RoboDK station: 29-6-1028.rdk

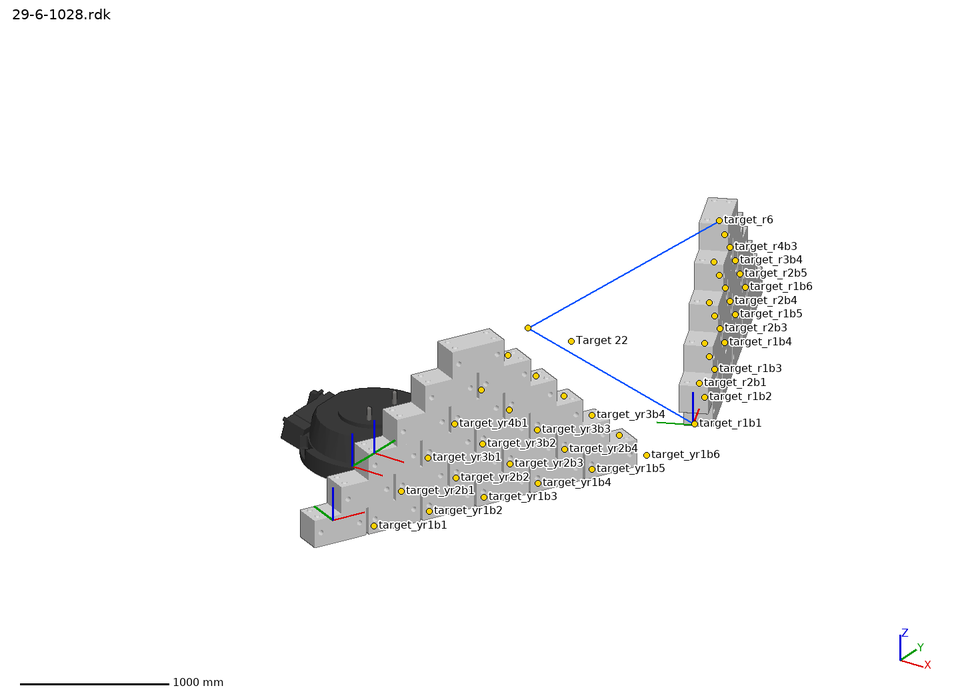
[picture v0: the station drawn from its stored meshes, robots at their saved joint values, targets as dots, program paths as lines]
Station 29-6-1028 (saved by RoboDK 5.4.1). Poses are relative to the parent item; angles as X-Y-Z fixed-axis rotations.
  - folder assets
    - object Floor at (0, 0, 0) mm, size 9000 x 9000 x 0 mm, geometry from Floor.sld
    - object Stairs_v1 at (-2520, 0, 0) mm, size 3922.2 x 7408.9 x 2302 mm, geometry from Stairs_v1.3ds
    - object Frame at (0, 0, 0) mm, size 2000 x 2500 x 199.8 mm, geometry from Frame.stp
  - frame KUKA KR 210-2 Base at (0, 0, 140) mm
    - robot KUKA KR 210-2: 6 axes, payload 210 kg, reach 2700 mm, repeatability 0.06 mm, weight 1267 kg
        joint limits [-185, -146, -119, -350, -125, -350] to [185, 0, 155, 350, 125, 350]; home [0, -128.166, 146.243, 0, -18.127, 0]; saved at [4.205, -124.52, 145.644, 6.755, -21.204, -6.343]
      - tool NEMO_ASM-v2, TCP at (50, 0, 430) mm, size 350 x 350 x 427.5 mm, geometry from NEMO_ASM-v2.stp
    - frame Table 1 at (2403.79, 306.78, 760.01) mm, rotated rx 0 ry 0 rz 115.9 deg
      - target target_r1b1 (Cartesian target) at (-6.3, -11.13, 11.37) mm, rotated rx -176.72 ry 88.61 rz 93.44 deg; joints [-0.522, -50.102, 99.56, 32.766, -52.796, -20.524] of KUKA KR 210-2
      - target target_r1b2 (Cartesian target) at (416.03, -12.09, 10.91) mm, rotated rx -158.93 ry 88.69 rz 112.47 deg; joints [-13.142, -53.707, 107.729, 17.568, -54.069, -9.744] of KUKA KR 210-2
      - target target_r1b3 (Cartesian target) at (839.45, -13.29, 13.06) mm, rotated rx 172.71 ry 89.07 rz 84.11 deg; joints [-27.608, -54.712, 110.113, -0.377, -54.484, 0.097] of KUKA KR 210-2
      - target target_r1b4 (Cartesian target) at (1261.96, -15.87, 12.69) mm, rotated rx 175.27 ry 88.55 rz 86.33 deg; joints [-41.947, -53.093, 105.958, -18.915, -52.906, 11.169] of KUKA KR 210-2
      - target target_r1b5 (Cartesian target) at (1681.19, -17.51, 17.53) mm, rotated rx 170.01 ry 89.31 rz 81.06 deg; joints [-54.307, -48.398, 95.994, -35.345, -52.576, 22.843] of KUKA KR 210-2
      - target target_r1b6 (Cartesian target) at (2102.3, -19.1, 19.95) mm, rotated rx -105.14 ry 89.86 rz 166.05 deg; joints [-64.353, -40.838, 79.979, -50.347, -51.856, 36.8] of KUKA KR 210-2
      - target target_r2b1 (Cartesian target) at (205.96, -10.53, 214.78) mm, rotated rx -150.39 ry 88.9 rz 120.14 deg; joints [-6.706, -59.689, 102.908, 28.081, -45.79, -19.523] of KUKA KR 210-2
      - target target_r2b2 (Cartesian target) at (625.98, -11.98, 212.77) mm, rotated rx -150.6 ry 88.91 rz 119.96 deg; joints [-20.566, -62.512, 108.17, 8.347, -45.007, -5.288] of KUKA KR 210-2
      - target target_r2b3 (Cartesian target) at (1050.36, -15.25, 215.86) mm, rotated rx -170.53 ry 89.44 rz 100.79 deg; joints [-34.887, -61.925, 107.233, -10.832, -45.265, 7.688] of KUKA KR 210-2
      - target target_r2b4 (Cartesian target) at (1470.51, -16.51, 217.48) mm, rotated rx -170.97 ry 89.43 rz 100.55 deg; joints [-48.227, -58.207, 100.325, -29.828, -45.582, 21.741] of KUKA KR 210-2
      - target target_r2b5 (Cartesian target) at (1894.14, -18.95, 219.85) mm, rotated rx -105.55 ry 89.86 rz 166.1 deg; joints [-59.529, -51.207, 87.402, -46.619, -46.767, 36.046] of KUKA KR 210-2
      - target target_r3b1 (Cartesian target) at (413.86, -11.7, 413.85) mm, rotated rx -150.56 ry 88.9 rz 120.16 deg; joints [-13.32, -67.987, 102.857, 22.975, -36.114, -18.141] of KUKA KR 210-2
      - target target_r3b2 (Cartesian target) at (838.41, -13.47, 414.6) mm, rotated rx -150.71 ry 88.91 rz 120.13 deg; joints [-27.82, -69.435, 105.015, -1.92, -34.642, 2.096] of KUKA KR 210-2
      - target target_r3b3 (Cartesian target) at (1261.16, -16.48, 417.6) mm, rotated rx -151.27 ry 88.9 rz 119.74 deg; joints [-41.958, -66.914, 100.942, -26.259, -35.938, 22.043] of KUKA KR 210-2
      - target target_r3b4 (Cartesian target) at (1682.3, -18.71, 421.05) mm, rotated rx -151.36 ry 88.9 rz 119.65 deg; joints [-54.347, -60.823, 90.919, -46.959, -39.086, 39.759] of KUKA KR 210-2
      - target target_r4b1 (Cartesian target) at (624.8, -11.3, 615.56) mm, rotated rx -147.6 ry 88.97 rz 122.93 deg; joints [-20.537, -74.49, 99.734, 14.025, -25.027, -12.111] of KUKA KR 210-2
      - target target_r4b2 (Cartesian target) at (1047.44, -13.61, 619.5) mm, rotated rx -147.6 ry 88.97 rz 122.95 deg; joints [-35.111, -73.887, 98.689, -20.611, -25.358, 19.191] of KUKA KR 210-2
      - target target_r4b3 (Cartesian target) at (1468.93, -16.18, 623.74) mm, rotated rx -140.39 ry 89.15 rz 130.98 deg; joints [-48.247, -69.156, 91.95, -45.556, -30.098, 41.709] of KUKA KR 210-2
      - target target_r5b1 (Cartesian target) at (833.72, -11.72, 817.94) mm, rotated rx -147.49 ry 88.97 rz 122.96 deg; joints [-27.81, -78.41, 93.338, -5.981, -14.13, 6.335] of KUKA KR 210-2
      - target target_r5b2 (Cartesian target) at (1256.88, -16.27, 822.3) mm, rotated rx -147.48 ry 88.97 rz 122.91 deg; joints [-42.054, -75.327, 89.185, -51.557, -20.3, 50.066] of KUKA KR 210-2
      - target target_r6 (Cartesian target) at (1047.28, -13.5, 1024.61) mm, rotated rx -147.4 ry 88.97 rz 122.91 deg; joints [-35.198, -79.421, 83.552, -70.3, -9.557, 70.464] of KUKA KR 210-2
      - object r6 at (1070, 0, 1000) mm, size 400 x 200 x 210 mm, geometry from brick_Origin.sld
      - object r1b1 at (0, 0, 0) mm, size 400 x 200 x 210 mm, geometry from brick_Origin.sld
        - object r1b2 at (420, 0, 0) mm, size 400 x 200 x 210 mm, geometry from brick_Origin.sld
          - object r1b3 at (420, 0, 0) mm, size 400 x 200 x 210 mm, geometry from brick_Origin.sld
            - object r1b4 at (420, 0, 0) mm, size 400 x 200 x 210 mm, geometry from brick_Origin.sld
              - object r1b5 at (420, 0, 0) mm, size 400 x 200 x 210 mm, geometry from brick_Origin.sld
                - object r1b6 at (420, 0, 0) mm, size 400 x 200 x 210 mm, geometry from brick_Origin.sld
      - object r2b1 at (210, 0, 200) mm, size 400 x 200 x 210 mm, geometry from brick_Origin.sld
        - object r2b2 at (420, 0, 0) mm, size 400 x 200 x 210 mm, geometry from brick_Origin.sld
          - object r2b3 at (420, 0, 0) mm, size 400 x 200 x 210 mm, geometry from brick_Origin.sld
            - object r2b4 at (420, 0, 0) mm, size 400 x 200 x 210 mm, geometry from brick_Origin.sld
              - object r2b5 at (420, 0, 0) mm, size 400 x 200 x 210 mm, geometry from brick_Origin.sld
      - object r3b1 at (420, 0, 400) mm, size 400 x 200 x 210 mm, geometry from brick_Origin.sld
        - object r3b2 at (420, 0, 0) mm, size 400 x 200 x 210 mm, geometry from brick_Origin.sld
          - object r3b3 at (420, 0, 0) mm, size 400 x 200 x 210 mm, geometry from brick_Origin.sld
            - object r3b4 at (420, 0, 0) mm, size 400 x 200 x 210 mm, geometry from brick_Origin.sld
      - object r4b1 at (640, 0, 600) mm, size 400 x 200 x 210 mm, geometry from brick_Origin.sld
        - object r4b2 at (420, 0, 0) mm, size 400 x 200 x 210 mm, geometry from brick_Origin.sld
          - object r4b3 at (420, 0, 0) mm, size 400 x 200 x 210 mm, geometry from brick_Origin.sld
      - object r5b1 at (860, 0, 800) mm, size 400 x 200 x 210 mm, geometry from brick_Origin.sld
        - object r5b2 at (420, 0, 0) mm, size 400 x 200 x 210 mm, geometry from brick_Origin.sld
      - target Target 22 (Cartesian target) at (65.85, 837.93, 530.04) mm, rotated rx 0 ry 89.95 rz -115.9 deg; joints [0, -103.679, 135.395, 0, -31.766, 0] of KUKA KR 210-2
    - frame Table 2 at (1260, -2281.06, 760) mm, rotated rx 0 ry 0 rz 65 deg
      - object r6 at (1070, 0, 1000) mm, size 400 x 200 x 210 mm, geometry from brick_Origin.sld
      - object r1b1 at (0, 0, 0) mm, size 400 x 200 x 210 mm, geometry from brick_Origin.sld
        - object r1b2 at (420, 0, 0) mm, size 400 x 200 x 210 mm, geometry from brick_Origin.sld
          - object r1b3 at (420, 0, 0) mm, size 400 x 200 x 210 mm, geometry from brick_Origin.sld
            - object r1b4 at (420, 0, 0) mm, size 400 x 200 x 210 mm, geometry from brick_Origin.sld
              - object r1b5 at (420, 0, 0) mm, size 400 x 200 x 210 mm, geometry from brick_Origin.sld
                - object r1b6 at (420, 0, 0) mm, size 400 x 200 x 210 mm, geometry from brick_Origin.sld
      - object r2b1 at (210, 0, 200) mm, size 400 x 200 x 210 mm, geometry from brick_Origin.sld
        - object r2b2 at (420, 0, 0) mm, size 400 x 200 x 210 mm, geometry from brick_Origin.sld
          - object r2b3 at (420, 0, 0) mm, size 400 x 200 x 210 mm, geometry from brick_Origin.sld
            - object r2b4 at (420, 0, 0) mm, size 400 x 200 x 210 mm, geometry from brick_Origin.sld
              - object r2b5 at (420, 0, 0) mm, size 400 x 200 x 210 mm, geometry from brick_Origin.sld
      - object r3b1 at (420, 0, 400) mm, size 400 x 200 x 210 mm, geometry from brick_Origin.sld
        - object r3b2 at (420, 0, 0) mm, size 400 x 200 x 210 mm, geometry from brick_Origin.sld
          - object r3b3 at (420, 0, 0) mm, size 400 x 200 x 210 mm, geometry from brick_Origin.sld
            - object r3b4 at (420, 0, 0) mm, size 400 x 200 x 210 mm, geometry from brick_Origin.sld
      - object r4b1 at (640, 0, 600) mm, size 400 x 200 x 210 mm, geometry from brick_Origin.sld
        - object r4b2 at (420, 0, 0) mm, size 400 x 200 x 210 mm, geometry from brick_Origin.sld
          - object r4b3 at (420, 0, 0) mm, size 400 x 200 x 210 mm, geometry from brick_Origin.sld
      - object r5b1 at (860, 0, 800) mm, size 400 x 200 x 210 mm, geometry from brick_Origin.sld
        - object r5b2 at (420, 0, 0) mm, size 400 x 200 x 210 mm, geometry from brick_Origin.sld
      - target target_yr1b1 (Cartesian target) at (191.06, -221.79, 6.64) mm, rotated rx 177.26 ry 87.95 rz 86.99 deg; joints [63.76, -40.183, 77.892, 54.102, -50.155, -39.985] of KUKA KR 210-2
      - target target_yr1b2 (Cartesian target) at (619.67, -222.93, 9.61) mm, rotated rx 176.38 ry 87.96 rz 87.14 deg; joints [53.941, -47.818, 94.114, 39.401, -51.283, -26.16] of KUKA KR 210-2
      - target target_yr1b3 (Cartesian target) at (1043.11, -221.89, 12.9) mm, rotated rx 177.38 ry 88.67 rz 88.48 deg; joints [41.815, -52.415, 104.57, 22.654, -52.993, -13.733] of KUKA KR 210-2
      - target target_yr1b4 (Cartesian target) at (1465.9, -221.29, 16.11) mm, rotated rx 177.17 ry 88.67 rz 88.44 deg; joints [27.869, -54.524, 108.938, 5.176, -53.196, -3.076] of KUKA KR 210-2
      - target target_yr1b5 (Cartesian target) at (1886.48, -221.45, 17.13) mm, rotated rx 176.96 ry 88.67 rz 88.39 deg; joints [13.646, -53.72, 107.063, -12.515, -52.663, 7.365] of KUKA KR 210-2
      - target target_yr1b6 (Cartesian target) at (2309.09, -219.38, 18.52) mm, rotated rx 176.64 ry 88.67 rz 88.34 deg; joints [0.644, -50.203, 99.231, -29.472, -51.504, 18.748] of KUKA KR 210-2
      - target target_yr2b1 (Cartesian target) at (402.62, -221.71, 211.66) mm, rotated rx 178.35 ry 88.63 rz 88.89 deg; joints [59.297, -50.26, 85.114, 51.802, -46.606, -40.211] of KUKA KR 210-2
      - target target_yr2b2 (Cartesian target) at (825.3, -222.42, 212.76) mm, rotated rx 178.46 ry 88.63 rz 88.87 deg; joints [48.158, -57.403, 98.507, 34.363, -45.074, -25.215] of KUKA KR 210-2
      - target target_yr2b3 (Cartesian target) at (1249.23, -222, 214.43) mm, rotated rx 178.17 ry 88.63 rz 88.9 deg; joints [34.991, -61.48, 105.821, 15.531, -44.015, -11.087] of KUKA KR 210-2
      - target target_yr2b4 (Cartesian target) at (1674.21, -220.18, 216.21) mm, rotated rx 177.61 ry 88.63 rz 88.91 deg; joints [20.733, -62.291, 107.138, -4.31, -43.561, 2.998] of KUKA KR 210-2
      - target target_yr2b5 (Cartesian target) at (2095.87, -220.1, 219.06) mm, rotated rx 177.64 ry 88.63 rz 88.88 deg; joints [6.849, -59.66, 102.184, -24.814, -43.859, 17.966] of KUKA KR 210-2
      - target target_yr3b1 (Cartesian target) at (610.67, -220.2, 414.28) mm, rotated rx 178.74 ry 88.63 rz 88.87 deg; joints [54.034, -59.853, 89.437, 49.893, -39.555, -41.737] of KUKA KR 210-2
      - target target_yr3b2 (Cartesian target) at (1034.81, -220.91, 414.61) mm, rotated rx 178.75 ry 88.36 rz 89.36 deg; joints [41.907, -66.176, 99.486, 31.068, -35.682, -25.596] of KUKA KR 210-2
      - target target_yr3b3 (Cartesian target) at (1458.98, -220.78, 416.7) mm, rotated rx 178.58 ry 88.45 rz 89.58 deg; joints [27.997, -68.982, 103.737, 7.264, -33.411, -6.004] of KUKA KR 210-2
      - target target_yr3b4 (Cartesian target) at (1883.7, -220.18, 418.97) mm, rotated rx -172.6 ry 88.43 rz 98.29 deg; joints [13.515, -67.866, 101.889, -19.226, -33.949, 16.046] of KUKA KR 210-2
      - target target_yr4b1 (Cartesian target) at (817.67, -220.56, 617.37) mm, rotated rx -168.2 ry 88.97 rz 101.69 deg; joints [48.227, -67.989, 90.381, 49.599, -31.018, -44.555] of KUKA KR 210-2
      - target target_yr4b2 (Cartesian target) at (1242.84, -220.85, 617.25) mm, rotated rx -168.58 ry 88.97 rz 101.73 deg; joints [35.042, -72.988, 97.499, 24.62, -25.54, -22.074] of KUKA KR 210-2
      - target target_yr4b3 (Cartesian target) at (1667.76, -220.3, 620.23) mm, rotated rx -168.88 ry 88.97 rz 101.82 deg; joints [20.711, -73.955, 98.642, -8.877, -23.928, 8.261] of KUKA KR 210-2
      - target target_yr5b1 (Cartesian target) at (1024.46, -220.23, 819.44) mm, rotated rx -168.91 ry 88.96 rz 101.03 deg; joints [41.993, -74.351, 87.969, 54.482, -20.962, -52.095] of KUKA KR 210-2
      - target target_yr5b2 (Cartesian target) at (1450.16, -219.75, 821.2) mm, rotated rx -167.72 ry 88.95 rz 102.56 deg; joints [28.009, -77.638, 92.1, 13.856, -13.818, -13.187] of KUKA KR 210-2
      - target target_yr6 (Cartesian target) at (1232.2, -220.04, 1026.38) mm, rotated rx -167.32 ry 88.95 rz 102.62 deg; joints [35.26, -78.462, 82.197, 75.378, -10.544, -74.722] of KUKA KR 210-2
    - frame Base at (0, -250.97, 0) mm
      - target Approach (Cartesian target) at (1266.25, 250.97, 1289.74) mm, rotated rx 0 ry 89.95 rz 0 deg; joints [0, -128.166, 146.243, 0, -18.127, 0] of KUKA KR 210-2
  - program Pick and place (10 instructions, listed below)
  - Python program Main (listed below)
  - program Prog3 (3 instructions, listed below)
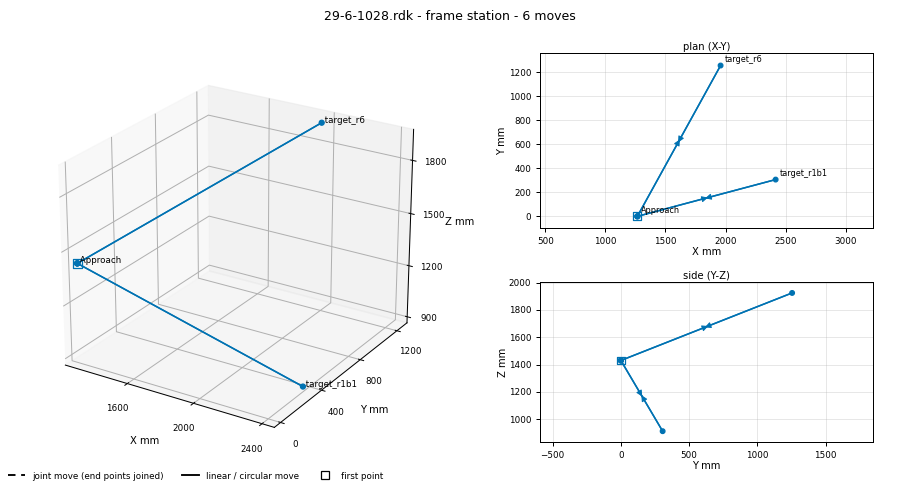
[picture p0: tool path of 29-6-1028.rdk in frame station, 6 of 6 moves have a stored position in this frame; points joined in program order, loops and branches not executed]

--- program Pick and place (robot KUKA KR 210-2) ---
  Set Frame: Table 1
  Set Tool: NEMO_ASM-v2
  Set speed (200.0 mm/s)
  MoveJ (Approach)
  MoveL (target_top) -> target target_r6
  MoveL (Approach)
  Set Ref.: Table 2
  MoveJ (Approach)
  MoveL (target_r1b1)
  MoveL (Approach)

--- Python program Main ---
# Type help("robodk.robolink") or help("robodk.robomath") for more information
# Press F5 to run the script
# Documentation: https://robodk.com/doc/en/RoboDK-API.html
# Reference:     https://robodk.com/doc/en/PythonAPI/robodk.html
# Note: It is not required to keep a copy of this file, your Python script is saved with your RDK project
from robodk import robolink    # RoboDK API
from robodk import robomath    # Robot toolbox

# The following 2 lines keep your code compatible with older versions or RoboDK:
from robodk import *      # RoboDK API
from robolink import *    # Robot toolbox

# Link to RoboDK
RDK = robolink.Robolink()
robot = RDK.Item('KUKA KR 210-2')
robot.setPoseFrame(robot.PoseFrame())
robot.setPoseTool(RDK.Item('NEMO_ASM-v2'))
robot.setAcceleration(600)

frame1 = RDK.Item('Table 1')
frame2 = RDK.Item('Table 2')
base = RDK.Item('Base')

speed_fast = 600
speed_slow = 200

pairList = [
    ['r6','yr1b1'],
    ['r5b2','yr1b2'],
    ['r5b1','yr1b3'],
    ['r4b3','yr1b4'],
    ['r4b2','yr1b5'],
    ['r4b1','yr1b6'],
    ['r3b4','yr2b1'],
    ['r3b3','yr2b2'],
    ['r3b2','yr2b3'],
    ['r3b1','yr2b4'],
    ['r2b5','yr2b5'],
    ['r2b4','yr3b1'],
    ['r2b3','yr3b2'],
    ['r2b2','yr3b3'],
    ['r2b1','yr3b4'],
    ['r1b6','yr4b1'],
    ['r1b5','yr4b2'],
    ['r1b4','yr4b3'],
    ['r1b3','yr5b1'],
    ['r1b2','yr5b2'],
    ['r1b1','yr6'],
]

def moveWithOffset(target_pose, offset):
    xyz_ref = target_pose.Pos()

    x = xyz_ref[0] + offset[0]
    y = xyz_ref[1] + offset[1]
    z = xyz_ref[2] + offset[2]

    target_pose.setPos([x,y,z])
    robot.MoveL(target_pose)
    return target_pose

def moveToBase():
    robot.setPoseFrame(base)

    target = RDK.Item('Approach')
    target_pose = target.Pose()
    robot.MoveL(target_pose)

def pickBrick(target_name):
    robot.setSpeed(speed_fast)

    target = RDK.Item(f'target_{target_name}')
    target_pose = target.Pose()

    approach_pose = moveWithOffset(target_pose, [0,300,0])
    robot.setSpeed(speed_slow)
    insert_pose = moveWithOffset(approach_pose, [0,-300,0])
    robot.setSpeed(speed_slow)
    lift_pose = moveWithOffset(insert_pose, [0,0,100])
    robot.setSpeed(speed_fast)
    safe_pose = moveWithOffset(lift_pose, [0,600,0])

def placeBrick(target_name):
    robot.setSpeed(speed_fast)

    target = RDK.Item(f'target_{target_name}')
    target_pose = target.Pose()

    approach_pose = moveWithOffset(target_pose, [0,300,100])
    robot.setSpeed(speed_slow)
    hovered_pos_insert = moveWithOffset(approach_pose, [0,-300,0])
    placed_pos = moveWithOffset(hovered_pos_insert, [0,0,-100])
    robot.setSpeed(speed_fast)
    safe_pos = moveWithOffset(placed_pos, [0,600,0])

def runMain(isFrameLeft):
    frameMain = frame1 if isFrameLeft else frame2
    frameAlter = frame2 if isFrameLeft else frame1

    if isFrameLeft:
        for i in pairList:
            robot.setPoseFrame(frameMain)
            pickBrick(i[0])
            moveToBase()
            robot.setPoseFrame(frameAlter)
            placeBrick(i[1])
            moveToBase()
    else:
        for i in reversed(pairList):
            robot.setPoseFrame(frameMain)
            pickBrick(i[1])
            moveToBase()
            robot.setPoseFrame(frameAlter)
            placeBrick(i[0])
            moveToBase()

    robot.RunInstruction('Program_Done')
    runMain(not isFrameLeft)

moveToBase()
runMain(isFrameLeft = True)
moveToBase()

--- program Prog3 (robot KUKA KR 210-2) ---
  Call Main
  Set speed (500.0 mm/s)
  Accurate (rounding -1 mm)
